// TwinCAT 3 PLC project txi_optics
// Title: lcls-plc-txi-optics
// Company: SLAC
// ProjectVersion: 0.2.0
// ProgramVersion: 3.1.4022.7
// libraries:
//   LCLS General, * (SLAC)
//   PMPS, * (SLAC - LCLS)
//   Tc2_ControllerToolbox, * (Beckhoff Automation GmbH)
//   Tc2_SerialCom, * (Beckhoff Automation GmbH)
//   Tc2_Standard, * (Beckhoff Automation GmbH)
//   Tc2_System, * (Beckhoff Automation GmbH)
//   Tc2_Utilities, * (Beckhoff Automation GmbH)
//   Tc3_Module, * (Beckhoff Automation GmbH)
//   lcls-twincat-motion,4.1.1,SLAC
//   lcls-twincat-optics,0.7.0,SLAC
// project tree:
//   GVLs/ GVL_COM_Buffers.TcGVL, GVL_M1K3.TcGVL, GVL_M1K3_Constants.TcGVL, GVL_M2K3.TcGVL, GVL_M2K3_Constants.TcGVL, GVL_PMPS.TcGVL, GVL_SerialIO.TcGVL
//   Version/ Global_Version.TcGVL
//   / PiezoDriver.TcTTO, PlcTask.TcTTO, SerialIO.TcTTO
//   POUs/ MAIN.TcPOU, PRG_1_PlcTask.TcPOU, PRG_2_PMPS_POST.TcPOU, PRG_MR1K3_SOMS.TcPOU, PRG_MR2K3_SOMS.TcPOU
//   POUs/Serial Comm/ PiezoSerial.TcPOU, P_Serial_Com.TcPOU
// real-time tasks:
//   TASK PlcTask: cycle T#10ms, priority 20, ADS port 350
//   TASK PiezoDriver: cycle T#1ms, priority 3, ADS port 351
//   TASK SerialIO: cycle T#2ms, priority 1, ADS port 352
// motion (NC):
//   TASK NC-Task 1 SAF: cycle T#2ms, priority 4, ADS port 501
//   TASK NC-Task 1 SVB: cycle T#10ms, priority 8, ADS port 511
//   AXIS M1K3-Yup (id 1)
//     General: UnitName=um
//     Dynamic: Acceleration=5050, Deceleration=5050, Jerk=5100500, DelayTime=0.008
//     Velo: Maximum=100
//     OtherSettings: AllowMotionCmdToSlave=true
//     encoder EncType=29
//       EncPara: ScaleFactorNumerator=1, ScaleFactorDenominator=1000, MaxCount=#xffffffff
//         SoftEndMinControl: Enable=true, Range=8900
//         SoftEndMaxControl: Enable=true, Range=122000
//         Inc: RefSoftSyncMask=#x0000ffff
//     drive DrvType=24
//       DrvPara: Inverse=true
//         Analog: VeloReferenz=500
//         TimeComp: TaskDelayCycles=1
//     controller CtrType=3
//       CtrPara: PriorControlFactor=1
//         PosDiffControl: Range=50, Time=0.2
//         PID: PosTn=0.005, PosIOutputLimit=0.0001, PosDOutputLimit=0, PosIDisableWhenMoving=true, DeadBandPosition=0.001
//         Observer: BandWidth=20
//   AXIS M1K3-Ydwn (id 2)
//     General: UnitName=um
//     Dynamic: Acceleration=5050, Deceleration=5050, Jerk=5100500, DelayTime=0.008
//     Velo: Maximum=100
//     OtherSettings: AllowMotionCmdToSlave=true
//     encoder EncType=29
//       EncPara: ScaleFactorNumerator=1, ScaleFactorDenominator=1000, MaxCount=#xffffffff
//         SoftEndMinControl: Enable=true, Range=8395
//         SoftEndMaxControl: Enable=true, Range=122000
//         Inc: RefSoftSyncMask=#x0000ffff
//     drive DrvType=24
//       DrvPara: Inverse=true
//         Analog: VeloReferenz=500
//         TimeComp: TaskDelayCycles=1
//     controller CtrType=3
//       CtrPara: PriorControlFactor=1
//         PosDiffControl: Range=50, Time=0.2
//         PID: PosTn=0.005, PosIOutputLimit=0.0001, PosDOutputLimit=0, PosIDisableWhenMoving=true, DeadBandPosition=0.001
//         Observer: BandWidth=20
//   AXIS M1K3-Xup (id 3)
//     General: UnitName=um
//     Dynamic: AccelerationMaximum=1000, DecelerationMaximum=1000, Acceleration=1000, Deceleration=1000, Jerk=5000, DelayTime=0.008
//     Velo: Maximum=300
//     OtherSettings: AllowMotionCmdToSlave=true
//     encoder EncType=29
//       EncPara: ScaleFactorNumerator=1, ScaleFactorDenominator=1000, MaxCount=#xffffffff
//         SoftEndMinControl: Enable=true, Range=20176
//         SoftEndMaxControl: Enable=true, Range=21576
//         Inc: RefSoftSyncMask=#x0000ffff
//     drive DrvType=24
//       DrvPara: Inverse=true
//         Analog: VeloReferenz=625
//         TimeComp: TaskDelayCycles=1
//     controller CtrType=3
//       CtrPara: PriorControlFactor=1
//         PosDiffControl: Range=50, Time=0.2
//         PID: PosTn=0.005, PosIOutputLimit=0.0001, PosDOutputLimit=0, PosIDisableWhenMoving=true, DeadBandPosition=0.001
//         Observer: BandWidth=20
//   AXIS M1K3-Xdwn (id 4)
//     General: UnitName=um
//     Dynamic: AccelerationMaximum=1000, DecelerationMaximum=1000, Acceleration=1000, Deceleration=1000, Jerk=5000, DelayTime=0.008
//     Velo: Maximum=300
//     OtherSettings: AllowMotionCmdToSlave=true
//     encoder EncType=29
//       EncPara: ScaleFactorNumerator=1, ScaleFactorDenominator=1000, MaxCount=#xffffffff
//         SoftEndMinControl: Enable=true, Range=21276
//         SoftEndMaxControl: Enable=true, Range=22876
//         Inc: RefSoftSyncMask=#x0000ffff
//     drive DrvType=24
//       Analog: VeloReferenz=625
//       TimeComp: TaskDelayCycles=1
//     controller CtrType=3
//       CtrPara: PriorControlFactor=1
//         PosDiffControl: Range=50, Time=0.2
//         PID: PosTn=0.005, PosIOutputLimit=0.0001, PosDOutputLimit=0, PosIDisableWhenMoving=true, DeadBandPosition=0.001
//         Observer: BandWidth=20
//   AXIS M1K3-Pitch (id 5)
//     General: UnitName=urad
//     Dynamic: Acceleration=64082, Deceleration=64082, Jerk=711156, DelayTime=0.008
//     Velo: Maximum=50
//     OtherSettings: AllowMotionCmdToSlave=true
//     encoder EncType=29
//       EncPara: ScaleFactorNumerator=0.00556, MaxCount=#xffffffff
//         SoftEndMinControl: Enable=true, Range=53575
//         SoftEndMaxControl: Enable=true, Range=54180
//         ActPosCorrection: Time=0.008
//         Inc: RefSoftSyncMask=#x0000ffff
//     drive DrvType=24
//       DrvPara: Inverse=true
//         Analog: VeloReferenz=550
//         TimeComp: TaskDelayCycles=1
//     controller CtrType=3
//       CtrPara: PriorControlFactor=1
//         PosDiffControl: Range=10, Time=0.2
//         PID: PosKp=9, PosTn=0.0006, PosTv=1.2e-05, PosIOutputLimit=0.0005, PosDOutputLimit=0.0035, AccKa=0.001, DeadBandPosition=0.1
//         Observer: BandWidth=20
//   AXIS Axis-None1 (id 11)
//     OtherSettings: AllowMotionCmdToSlave=true
//     encoder EncType=1
//     drive DrvType=5
//       Analog: ScaleFactorActTorque=0.1
//     controller CtrType=1
//       CtrPara: PriorControlFactor=1
//         Observer: BandWidth=20
//   AXIS M2K3-Yup (id 6)
//     General: UnitName=um
//     Dynamic: Acceleration=5050, Deceleration=5050, Jerk=5100500, DelayTime=0.008
//     Velo: Maximum=100
//     TargetPosControl: Range=0.05, Time=0.01
//     OtherSettings: AllowMotionCmdToSlave=true
//     encoder EncType=29
//       EncPara: ScaleFactorNumerator=1, ScaleFactorDenominator=1000, MaxCount=#xffffffff
//         SoftEndMinControl: Enable=true, Range=7250
//         SoftEndMaxControl: Enable=true, Range=115658
//         Inc: RefSoftSyncMask=#x0000ffff
//     drive DrvType=24
//       DrvPara: Inverse=true
//         Analog: VeloReferenz=500
//         TimeComp: TaskDelayCycles=1
//     controller CtrType=3
//       CtrPara: PriorControlFactor=1
//         PosDiffControl: Range=50, Time=0.2
//         PID: PosTn=0.005, PosIOutputLimit=0.0001, PosDOutputLimit=0, PosIDisableWhenMoving=true, DeadBandPosition=0.001
//         Observer: BandWidth=20
//   AXIS M2K3-Ydwn (id 7)
//     General: UnitName=um
//     Dynamic: Acceleration=5050, Deceleration=5050, Jerk=5100500, DelayTime=0.008
//     Velo: Maximum=100
//     TargetPosControl: Range=0.05, Time=0.01
//     OtherSettings: AllowMotionCmdToSlave=true
//     encoder EncType=29
//       EncPara: ScaleFactorNumerator=1, ScaleFactorDenominator=1000, MaxCount=#xffffffff
//         SoftEndMinControl: Enable=true, Range=9960
//         SoftEndMaxControl: Enable=true, Range=118260
//         Inc: RefSoftSyncMask=#x0000ffff
//     drive DrvType=24
//       DrvPara: Inverse=true
//         Analog: VeloReferenz=500
//         TimeComp: TaskDelayCycles=1
//     controller CtrType=3
//       CtrPara: PriorControlFactor=1
//         PosDiffControl: Range=50, Time=0.2
//         PID: PosTn=0.005, PosIOutputLimit=0.0001, PosDOutputLimit=0, PosIDisableWhenMoving=true, DeadBandPosition=0.001
//         Observer: BandWidth=20
//   AXIS M2K3-Xup (id 8)
//     General: UnitName=um
//     Dynamic: AccelerationMaximum=1000, DecelerationMaximum=1000, Acceleration=1000, Deceleration=1000, Jerk=5000, DelayTime=0.008
//     Velo: Maximum=150
//     TargetPosControl: Range=0.05, Time=0.01
//     OtherSettings: AllowMotionCmdToSlave=true
//     encoder EncType=29
//       EncPara: ScaleFactorNumerator=1, ScaleFactorDenominator=1000, MaxCount=#xffffffff
//         SoftEndMinControl: Enable=true, Range=19294
//         SoftEndMaxControl: Enable=true, Range=20694
//         Inc: RefSoftSyncMask=#x0000ffff
//     drive DrvType=24
//       DrvPara: Inverse=true
//         Analog: VeloReferenz=625
//         TimeComp: TaskDelayCycles=1
//     controller CtrType=3
//       CtrPara: PriorControlFactor=1
//         PosDiffControl: Range=50, Time=0.2
//         PID: PosTn=0.005, PosIOutputLimit=0.0001, PosDOutputLimit=0, PosIDisableWhenMoving=true, DeadBandPosition=0.001
//         Observer: BandWidth=20
//   AXIS M2K3-Xdwn (id 9)
//     General: UnitName=um
//     Dynamic: AccelerationMaximum=1000, DecelerationMaximum=1000, Acceleration=1000, Deceleration=1000, Jerk=5000, DelayTime=0.008
//     Velo: Maximum=150
//     TargetPosControl: Range=0.05, Time=0.01
//     OtherSettings: AllowMotionCmdToSlave=true
//     encoder EncType=29
//       EncPara: ScaleFactorNumerator=1, ScaleFactorDenominator=1000, MaxCount=#xffffffff
//         SoftEndMinControl: Enable=true, Range=18074
//         SoftEndMaxControl: Enable=true, Range=19674
//         Inc: RefSoftSyncMask=#x0000ffff
//     drive DrvType=24
//       Analog: VeloReferenz=625
//       TimeComp: TaskDelayCycles=1
//     controller CtrType=3
//       CtrPara: PriorControlFactor=1
//         PosDiffControl: Range=50, Time=0.2
//         PID: PosTn=0.005, PosIOutputLimit=0.0001, PosDOutputLimit=0, PosIDisableWhenMoving=true, DeadBandPosition=0.001
//         Observer: BandWidth=20
//   AXIS M2K3-Pitch (id 10)
//     General: UnitName=urad
//     Dynamic: Acceleration=64082, Deceleration=64082, Jerk=711156, DelayTime=0.008
//     Velo: SlowManual=10, FastManual=30, Maximum=50
//     TargetPosControl: Range=0.1, Time=0.01
//     PEHControl: Time=7
//     OtherSettings: AllowMotionCmdToSlave=true
//     encoder EncType=29
//       EncPara: ScaleFactorNumerator=0.00556, MaxCount=#xffffffff
//         FilterTime: TPos=0.05
//         SoftEndMinControl: Enable=true, Range=57450
//         SoftEndMaxControl: Enable=true, Range=59067
//         ActPosCorrection: Time=0.008
//         Inc: RefSoftSyncMask=#x0000ffff
//     drive DrvType=24
//       DrvPara: Inverse=true
//         Analog: VeloReferenz=550
//         TimeComp: TaskDelayCycles=1
//     controller CtrType=3
//       CtrPara: PriorControlFactor=1
//         PosDiffControl: Range=10, Time=0.2
//         PID: PosKp=9, PosTn=0.0006, PosTv=1.2e-05, PosIOutputLimit=0.0005, PosDOutputLimit=0.0035, AccKa=0.001, DeadBandPosition=0.001
//         Observer: BandWidth=20
//   AXIS Axis-None2 (id 12)
//     OtherSettings: AllowMotionCmdToSlave=true
//     encoder EncType=1
//     drive DrvType=5
//       Analog: ScaleFactorActTorque=0.1
//     controller CtrType=1
//       CtrPara: PriorControlFactor=1
//         Observer: BandWidth=20
// I/O:
//   DEVICE Device 1 (EtherCAT), AmsNetId 172.21.88.54.2.1
//     Term 1 (EK1200) [EK1200-5000 EtherCAT Power supply (2A E-Bus)]
//       PMPS_FFO [EL2202 2Ch. Dig. Output 24V, 0.5A]
//       Term 3 (EL6070)
//       PMPS_PRE [EL6695 EtherCAT Bridge terminal (Primary)]
//       Term 6 (EK1122) [EK1122 2 port EtherCAT junction]
//         EK1100_M1K3 [EK1100 EtherCAT Coupler (2A E-Bus)]
//           Term 8 (EL9410)
//           EL7047_M1K3_Yup [EL7047 1Ch. Stepper motor output stage (50V, 5A)]
//           EL7047_M1K3_Ydwn [EL7047 1Ch. Stepper motor output stage (50V, 5A)]
//           EL7047_M1K3_Xup [EL7047 1Ch. Stepper motor output stage (50V, 5A)]
//           EL7047_M1K3_Xdwn [EL7047 1Ch. Stepper motor output stage (50V, 5A)]
//           EL7047_M1K3_PitchCoarse [EL7047 1Ch. Stepper motor output stage (50V, 5A)]
//           EL5042_M1K3_Yupdwn [EL5042 2Ch. BiSS-C Encoder]
//           EL5042_M1K3_Xupdwn
//           EL5042_M1K3_Pitch [EL5042 2Ch. BiSS-C Encoder]
//           EL6001_M1K3_PitchFine [EL6001 Interface (RS232)]
//           EL3054_M1K3_FWM_PRSM [EL3054 4Ch. Ana. Input 4-20mA]
//           Term 19 (EL3202-0010)
//           Term 20 (EL3202-0010)
//           EL1004_M1K3_STO [EL1004 4Ch. Dig. Input 24V, 3ms]
//           EL2004_M1K3_VCV [EL2004 4Ch. Dig. Output 24V, 0.5A]
//           Term 36 (EL9011) [EL9011 End Terminal]
//         EK1100_M2K3 [EK1100 EtherCAT Coupler (2A E-Bus)]
//           Term 22 (EL9410) [EL9410 E-Bus Power Supplier  (Diagnostics)]
//           EL7047_M2K3_Yup [EL7047 1Ch. Stepper motor output stage (50V, 5A)]
//           EL7047_M2K3_Ydwn [EL7047 1Ch. Stepper motor output stage (50V, 5A)]
//           EL7047_M2K3_Xup [EL7047 1Ch. Stepper motor output stage (50V, 5A)]
//           EL7047_M2K3_Xdwn [EL7047 1Ch. Stepper motor output stage (50V, 5A)]
//           EL7047_M2K3_PitchCoarse [EL7047 1Ch. Stepper motor output stage (50V, 5A)]
//           EL5042_M2K3_Yupdwn [EL5042 2Ch. BiSS-C Encoder]
//           EL5042_M2K3_Xupdwn [EL5042 2Ch. BiSS-C Encoder]
//           EL5042_M2K3_Pitch [EL5042 2Ch. BiSS-C Encoder]
//           EL6001_M2K3_PitchFine [EL6001 Interface (RS232)]
//           EL3054_M2K3_FWM_PRSM [EL3054 4Ch. Ana. Input 4-20mA]
//           Term 33 (EL3202-0010) [EL3202-0010 2Ch. Ana. Input PT100 (RTD), High Precision]
//           Term 34 (EL3202-0010) [EL3202-0010 2Ch. Ana. Input PT100 (RTD), High Precision]
//           EL1004_M2K3_STO [EL1004 4Ch. Dig. Input 24V, 3ms]
//           EL2004_M2K3_VCV [EL2004 4Ch. Dig. Output 24V, 0.5A]
//           Term 37 (EL9011) [EL9011 End Terminal]
//       Term 35 (EK1122) [EK1122 2 port EtherCAT junction]
//       Term 38 (EL9011)
// variable links:
//   (this object) <-> Device 1 (EtherCAT)/Term 1 (EK1200)/Term 6 (EK1122)/EK1100_M1K3/EL5042_M1K3_Yupdwn
//     Enc/Inputs/In/nComState @bit 1 <-> WcState/InputToggle
//     Enc/Inputs/In/nComState <-> WcState/WcState
//     Enc/Inputs/In/nDataIn1 <-> FB Inputs Channel 1/Position
//     Enc/Inputs/In/nDataIn1 <-> FB Inputs Channel 2/Position
//     Enc/Inputs/In/nState1 @bit 12 <-> FB Inputs Channel 1/Status/Diag
//     Enc/Inputs/In/nState1 @bit 12 <-> FB Inputs Channel 2/Status/Diag
//     Enc/Inputs/In/nState1 @bit 1 <-> FB Inputs Channel 1/Status/Error
//     Enc/Inputs/In/nState1 @bit 1 <-> FB Inputs Channel 2/Status/Error
//     Enc/Inputs/In/nState1 @bit 14 <-> FB Inputs Channel 1/Status/Input cycle counter
//     Enc/Inputs/In/nState1 @bit 14 <-> FB Inputs Channel 2/Status/Input cycle counter
//     Enc/Inputs/In/nState1 @bit 2 <-> FB Inputs Channel 1/Status/Ready
//     Enc/Inputs/In/nState1 @bit 2 <-> FB Inputs Channel 2/Status/Ready
//     Enc/Inputs/In/nState1 @bit 13 <-> FB Inputs Channel 1/Status/TxPDO State
//     Enc/Inputs/In/nState1 @bit 13 <-> FB Inputs Channel 2/Status/TxPDO State
//     Enc/Inputs/In/nState1 <-> FB Inputs Channel 1/Status/Warning
//     Enc/Inputs/In/nState1 <-> FB Inputs Channel 2/Status/Warning
//   (this object) <-> Device 1 (EtherCAT)/Term 1 (EK1200)/Term 6 (EK1122)/EK1100_M1K3/EL7047_M1K3_Yup
//     Drive/Inputs/In/nState1 @bit 3 <-> STM Status/Status/Error
//     Drive/Inputs/In/nState1 @bit 7 <-> STM Status/Status/Motor stall
//     Drive/Inputs/In/nState1 @bit 5 <-> STM Status/Status/Moving negative
//     Drive/Inputs/In/nState1 @bit 4 <-> STM Status/Status/Moving positive
//     Drive/Inputs/In/nState1 @bit 1 <-> STM Status/Status/Ready
//     Drive/Inputs/In/nState1 <-> STM Status/Status/Ready to enable
//     Drive/Inputs/In/nState1 @bit 6 <-> STM Status/Status/Torque reduced
//     Drive/Inputs/In/nState1 @bit 2 <-> STM Status/Status/Warning
//     Drive/Inputs/In/nState2 @bit 3 <-> STM Status/Status/Digital input 1
//     Drive/Inputs/In/nState2 @bit 4 <-> STM Status/Status/Digital input 2
//     Drive/Inputs/In/nState2 @bit 5 <-> STM Status/Status/Sync error
//     Drive/Inputs/In/nState2 @bit 7 <-> STM Status/Status/TxPDO Toggle
//     Drive/Inputs/In/nState4 @bit 1 <-> WcState/InputToggle
//     Drive/Inputs/In/nState4 <-> WcState/WcState
//     Drive/Outputs/Out/nCtrl1 <-> STM Control/Control/Enable
//     Drive/Outputs/Out/nCtrl1 @bit 2 <-> STM Control/Control/Reduce torque
//     Drive/Outputs/Out/nCtrl1 @bit 1 <-> STM Control/Control/Reset
//     Drive/Outputs/Out/nCtrl2 @bit 3 <-> STM Control/Control/Digital output 1
//     Drive/Outputs/Out/nDataOut2[0] <-> STM Velocity/Velocity
//   (this object) <-> Device 1 (EtherCAT)/Term 1 (EK1200)/Term 6 (EK1122)/EK1100_M1K3/EL7047_M1K3_Ydwn
//     Drive/Inputs/In/nState1 @bit 3 <-> STM Status/Status/Error
//     Drive/Inputs/In/nState1 @bit 7 <-> STM Status/Status/Motor stall
//     Drive/Inputs/In/nState1 @bit 5 <-> STM Status/Status/Moving negative
//     Drive/Inputs/In/nState1 @bit 4 <-> STM Status/Status/Moving positive
//     Drive/Inputs/In/nState1 @bit 1 <-> STM Status/Status/Ready
//     Drive/Inputs/In/nState1 <-> STM Status/Status/Ready to enable
//     Drive/Inputs/In/nState1 @bit 6 <-> STM Status/Status/Torque reduced
//     Drive/Inputs/In/nState1 @bit 2 <-> STM Status/Status/Warning
//     Drive/Inputs/In/nState2 @bit 3 <-> STM Status/Status/Digital input 1
//     Drive/Inputs/In/nState2 @bit 4 <-> STM Status/Status/Digital input 2
//     Drive/Inputs/In/nState2 @bit 5 <-> STM Status/Status/Sync error
//     Drive/Inputs/In/nState2 @bit 7 <-> STM Status/Status/TxPDO Toggle
//     Drive/Inputs/In/nState4 @bit 1 <-> WcState/InputToggle
//     Drive/Inputs/In/nState4 <-> WcState/WcState
//     Drive/Outputs/Out/nCtrl1 <-> STM Control/Control/Enable
//     Drive/Outputs/Out/nCtrl1 @bit 2 <-> STM Control/Control/Reduce torque
//     Drive/Outputs/Out/nCtrl1 @bit 1 <-> STM Control/Control/Reset
//     Drive/Outputs/Out/nCtrl2 @bit 3 <-> STM Control/Control/Digital output 1
//     Drive/Outputs/Out/nDataOut2[0] <-> STM Velocity/Velocity
//   (this object) <-> Device 1 (EtherCAT)/Term 1 (EK1200)/Term 6 (EK1122)/EK1100_M1K3/EL5042_M1K3_Xupdwn
//     Enc/Inputs/In/nComState @bit 1 <-> WcState/InputToggle
//     Enc/Inputs/In/nComState <-> WcState/WcState
//     Enc/Inputs/In/nDataIn1 <-> FB Inputs Channel 1/Position
//     Enc/Inputs/In/nDataIn1 <-> FB Inputs Channel 2/Position
//     Enc/Inputs/In/nState1 @bit 12 <-> FB Inputs Channel 1/Status/Diag
//     Enc/Inputs/In/nState1 @bit 12 <-> FB Inputs Channel 2/Status/Diag
//     Enc/Inputs/In/nState1 @bit 1 <-> FB Inputs Channel 1/Status/Error
//     Enc/Inputs/In/nState1 @bit 1 <-> FB Inputs Channel 2/Status/Error
//     Enc/Inputs/In/nState1 @bit 14 <-> FB Inputs Channel 1/Status/Input cycle counter
//     Enc/Inputs/In/nState1 @bit 14 <-> FB Inputs Channel 2/Status/Input cycle counter
//     Enc/Inputs/In/nState1 @bit 2 <-> FB Inputs Channel 1/Status/Ready
//     Enc/Inputs/In/nState1 @bit 2 <-> FB Inputs Channel 2/Status/Ready
//     Enc/Inputs/In/nState1 @bit 13 <-> FB Inputs Channel 1/Status/TxPDO State
//     Enc/Inputs/In/nState1 @bit 13 <-> FB Inputs Channel 2/Status/TxPDO State
//     Enc/Inputs/In/nState1 <-> FB Inputs Channel 1/Status/Warning
//     Enc/Inputs/In/nState1 <-> FB Inputs Channel 2/Status/Warning
//   (this object) <-> Device 1 (EtherCAT)/Term 1 (EK1200)/Term 6 (EK1122)/EK1100_M1K3/EL7047_M1K3_Xup
//     Drive/Inputs/In/nState1 @bit 3 <-> STM Status/Status/Error
//     Drive/Inputs/In/nState1 @bit 7 <-> STM Status/Status/Motor stall
//     Drive/Inputs/In/nState1 @bit 5 <-> STM Status/Status/Moving negative
//     Drive/Inputs/In/nState1 @bit 4 <-> STM Status/Status/Moving positive
//     Drive/Inputs/In/nState1 @bit 1 <-> STM Status/Status/Ready
//     Drive/Inputs/In/nState1 <-> STM Status/Status/Ready to enable
//     Drive/Inputs/In/nState1 @bit 6 <-> STM Status/Status/Torque reduced
//     Drive/Inputs/In/nState1 @bit 2 <-> STM Status/Status/Warning
//     Drive/Inputs/In/nState2 @bit 3 <-> STM Status/Status/Digital input 1
//     Drive/Inputs/In/nState2 @bit 4 <-> STM Status/Status/Digital input 2
//     Drive/Inputs/In/nState2 @bit 5 <-> STM Status/Status/Sync error
//     Drive/Inputs/In/nState2 @bit 7 <-> STM Status/Status/TxPDO Toggle
//     Drive/Inputs/In/nState4 @bit 1 <-> WcState/InputToggle
//     Drive/Inputs/In/nState4 <-> WcState/WcState
//     Drive/Outputs/Out/nCtrl1 <-> STM Control/Control/Enable
//     Drive/Outputs/Out/nCtrl1 @bit 2 <-> STM Control/Control/Reduce torque
//     Drive/Outputs/Out/nCtrl1 @bit 1 <-> STM Control/Control/Reset
//     Drive/Outputs/Out/nCtrl2 @bit 3 <-> STM Control/Control/Digital output 1
//     Drive/Outputs/Out/nDataOut2[0] <-> STM Velocity/Velocity
//   (this object) <-> Device 1 (EtherCAT)/Term 1 (EK1200)/Term 6 (EK1122)/EK1100_M1K3/EL7047_M1K3_Xdwn
//     Drive/Inputs/In/nState1 @bit 3 <-> STM Status/Status/Error
//     Drive/Inputs/In/nState1 @bit 7 <-> STM Status/Status/Motor stall
//     Drive/Inputs/In/nState1 @bit 5 <-> STM Status/Status/Moving negative
//     Drive/Inputs/In/nState1 @bit 4 <-> STM Status/Status/Moving positive
//     Drive/Inputs/In/nState1 @bit 1 <-> STM Status/Status/Ready
//     Drive/Inputs/In/nState1 <-> STM Status/Status/Ready to enable
//     Drive/Inputs/In/nState1 @bit 6 <-> STM Status/Status/Torque reduced
//     Drive/Inputs/In/nState1 @bit 2 <-> STM Status/Status/Warning
//     Drive/Inputs/In/nState2 @bit 3 <-> STM Status/Status/Digital input 1
//     Drive/Inputs/In/nState2 @bit 4 <-> STM Status/Status/Digital input 2
//     Drive/Inputs/In/nState2 @bit 5 <-> STM Status/Status/Sync error
//     Drive/Inputs/In/nState2 @bit 7 <-> STM Status/Status/TxPDO Toggle
//     Drive/Inputs/In/nState4 @bit 1 <-> WcState/InputToggle
//     Drive/Inputs/In/nState4 <-> WcState/WcState
//     Drive/Outputs/Out/nCtrl1 <-> STM Control/Control/Enable
//     Drive/Outputs/Out/nCtrl1 @bit 2 <-> STM Control/Control/Reduce torque
//     Drive/Outputs/Out/nCtrl1 @bit 1 <-> STM Control/Control/Reset
//     Drive/Outputs/Out/nCtrl2 @bit 3 <-> STM Control/Control/Digital output 1
//     Drive/Outputs/Out/nDataOut2[0] <-> STM Velocity/Velocity
//   (this object) <-> Device 1 (EtherCAT)/Term 1 (EK1200)/Term 6 (EK1122)/EK1100_M1K3/EL5042_M1K3_Pitch
//     Enc/Inputs/In/nComState @bit 1 <-> WcState/InputToggle
//     Enc/Inputs/In/nComState <-> WcState/WcState
//     Enc/Inputs/In/nDataIn1 <-> FB Inputs Channel 1/Position
//     Enc/Inputs/In/nState1 @bit 12 <-> FB Inputs Channel 1/Status/Diag
//     Enc/Inputs/In/nState1 @bit 1 <-> FB Inputs Channel 1/Status/Error
//     Enc/Inputs/In/nState1 @bit 14 <-> FB Inputs Channel 1/Status/Input cycle counter
//     Enc/Inputs/In/nState1 @bit 2 <-> FB Inputs Channel 1/Status/Ready
//     Enc/Inputs/In/nState1 @bit 13 <-> FB Inputs Channel 1/Status/TxPDO State
//     Enc/Inputs/In/nState1 <-> FB Inputs Channel 1/Status/Warning
//   (this object) <-> Device 1 (EtherCAT)/Term 1 (EK1200)/Term 6 (EK1122)/EK1100_M1K3/EL7047_M1K3_PitchCoarse
//     Drive/Inputs/In/nState1 @bit 3 <-> STM Status/Status/Error
//     Drive/Inputs/In/nState1 @bit 7 <-> STM Status/Status/Motor stall
//     Drive/Inputs/In/nState1 @bit 5 <-> STM Status/Status/Moving negative
//     Drive/Inputs/In/nState1 @bit 4 <-> STM Status/Status/Moving positive
//     Drive/Inputs/In/nState1 @bit 1 <-> STM Status/Status/Ready
//     Drive/Inputs/In/nState1 <-> STM Status/Status/Ready to enable
//     Drive/Inputs/In/nState1 @bit 6 <-> STM Status/Status/Torque reduced
//     Drive/Inputs/In/nState1 @bit 2 <-> STM Status/Status/Warning
//     Drive/Inputs/In/nState2 @bit 3 <-> STM Status/Status/Digital input 1
//     Drive/Inputs/In/nState2 @bit 4 <-> STM Status/Status/Digital input 2
//     Drive/Inputs/In/nState2 @bit 5 <-> STM Status/Status/Sync error
//     Drive/Inputs/In/nState2 @bit 7 <-> STM Status/Status/TxPDO Toggle
//     Drive/Inputs/In/nState4 @bit 1 <-> WcState/InputToggle
//     Drive/Inputs/In/nState4 <-> WcState/WcState
//     Drive/Outputs/Out/nCtrl1 <-> STM Control/Control/Enable
//     Drive/Outputs/Out/nCtrl1 @bit 2 <-> STM Control/Control/Reduce torque
//     Drive/Outputs/Out/nCtrl1 @bit 1 <-> STM Control/Control/Reset
//     Drive/Outputs/Out/nCtrl2 @bit 3 <-> STM Control/Control/Digital output 1
//     Drive/Outputs/Out/nDataOut2[0] <-> STM Velocity/Velocity
//   (this object) <-> Device 1 (EtherCAT)/Term 1 (EK1200)/Term 6 (EK1122)/EK1100_M2K3/EL5042_M2K3_Yupdwn
//     Enc/Inputs/In/nComState @bit 1 <-> WcState/InputToggle
//     Enc/Inputs/In/nComState <-> WcState/WcState
//     Enc/Inputs/In/nDataIn1 <-> FB Inputs Channel 1/Position
//     Enc/Inputs/In/nDataIn1 <-> FB Inputs Channel 2/Position
//     Enc/Inputs/In/nState1 @bit 12 <-> FB Inputs Channel 1/Status/Diag
//     Enc/Inputs/In/nState1 @bit 12 <-> FB Inputs Channel 2/Status/Diag
//     Enc/Inputs/In/nState1 @bit 1 <-> FB Inputs Channel 1/Status/Error
//     Enc/Inputs/In/nState1 @bit 1 <-> FB Inputs Channel 2/Status/Error
//     Enc/Inputs/In/nState1 @bit 14 <-> FB Inputs Channel 1/Status/Input cycle counter
//     Enc/Inputs/In/nState1 @bit 14 <-> FB Inputs Channel 2/Status/Input cycle counter
//     Enc/Inputs/In/nState1 @bit 2 <-> FB Inputs Channel 1/Status/Ready
//     Enc/Inputs/In/nState1 @bit 2 <-> FB Inputs Channel 2/Status/Ready
//     Enc/Inputs/In/nState1 @bit 13 <-> FB Inputs Channel 1/Status/TxPDO State
//     Enc/Inputs/In/nState1 @bit 13 <-> FB Inputs Channel 2/Status/TxPDO State
//     Enc/Inputs/In/nState1 <-> FB Inputs Channel 1/Status/Warning
//     Enc/Inputs/In/nState1 <-> FB Inputs Channel 2/Status/Warning
//   (this object) <-> Device 1 (EtherCAT)/Term 1 (EK1200)/Term 6 (EK1122)/EK1100_M2K3/EL7047_M2K3_Yup
//     Drive/Inputs/In/nState1 @bit 3 <-> STM Status/Status/Error
//     Drive/Inputs/In/nState1 @bit 7 <-> STM Status/Status/Motor stall
//     Drive/Inputs/In/nState1 @bit 5 <-> STM Status/Status/Moving negative
//     Drive/Inputs/In/nState1 @bit 4 <-> STM Status/Status/Moving positive
//     Drive/Inputs/In/nState1 @bit 1 <-> STM Status/Status/Ready
//     Drive/Inputs/In/nState1 <-> STM Status/Status/Ready to enable
//     Drive/Inputs/In/nState1 @bit 6 <-> STM Status/Status/Torque reduced
//     Drive/Inputs/In/nState1 @bit 2 <-> STM Status/Status/Warning
//     Drive/Inputs/In/nState2 @bit 3 <-> STM Status/Status/Digital input 1
//     Drive/Inputs/In/nState2 @bit 4 <-> STM Status/Status/Digital input 2
//     Drive/Inputs/In/nState2 @bit 5 <-> STM Status/Status/Sync error
//     Drive/Inputs/In/nState2 @bit 7 <-> STM Status/Status/TxPDO Toggle
//     Drive/Inputs/In/nState4 @bit 1 <-> WcState/InputToggle
//     Drive/Inputs/In/nState4 <-> WcState/WcState
//     Drive/Outputs/Out/nCtrl1 <-> STM Control/Control/Enable
//     Drive/Outputs/Out/nCtrl1 @bit 2 <-> STM Control/Control/Reduce torque
//     Drive/Outputs/Out/nCtrl1 @bit 1 <-> STM Control/Control/Reset
//     Drive/Outputs/Out/nCtrl2 @bit 3 <-> STM Control/Control/Digital output 1
//     Drive/Outputs/Out/nDataOut2[0] <-> STM Velocity/Velocity
//   (this object) <-> Device 1 (EtherCAT)/Term 1 (EK1200)/Term 6 (EK1122)/EK1100_M2K3/EL7047_M2K3_Ydwn
//     Drive/Inputs/In/nState1 @bit 3 <-> STM Status/Status/Error
//     Drive/Inputs/In/nState1 @bit 7 <-> STM Status/Status/Motor stall
//     Drive/Inputs/In/nState1 @bit 5 <-> STM Status/Status/Moving negative
//     Drive/Inputs/In/nState1 @bit 4 <-> STM Status/Status/Moving positive
//     Drive/Inputs/In/nState1 @bit 1 <-> STM Status/Status/Ready
//     Drive/Inputs/In/nState1 <-> STM Status/Status/Ready to enable
//     Drive/Inputs/In/nState1 @bit 6 <-> STM Status/Status/Torque reduced
//     Drive/Inputs/In/nState1 @bit 2 <-> STM Status/Status/Warning
//     Drive/Inputs/In/nState2 @bit 3 <-> STM Status/Status/Digital input 1
//     Drive/Inputs/In/nState2 @bit 4 <-> STM Status/Status/Digital input 2
//     Drive/Inputs/In/nState2 @bit 5 <-> STM Status/Status/Sync error
//     Drive/Inputs/In/nState2 @bit 7 <-> STM Status/Status/TxPDO Toggle
//     Drive/Inputs/In/nState4 @bit 1 <-> WcState/InputToggle
//     Drive/Inputs/In/nState4 <-> WcState/WcState
//     Drive/Outputs/Out/nCtrl1 <-> STM Control/Control/Enable
//     Drive/Outputs/Out/nCtrl1 @bit 2 <-> STM Control/Control/Reduce torque
//     Drive/Outputs/Out/nCtrl1 @bit 1 <-> STM Control/Control/Reset
//     Drive/Outputs/Out/nCtrl2 @bit 3 <-> STM Control/Control/Digital output 1
//     Drive/Outputs/Out/nDataOut2[0] <-> STM Velocity/Velocity
//   (this object) <-> Device 1 (EtherCAT)/Term 1 (EK1200)/Term 6 (EK1122)/EK1100_M2K3/EL5042_M2K3_Xupdwn
//     Enc/Inputs/In/nComState @bit 1 <-> WcState/InputToggle
//     Enc/Inputs/In/nComState <-> WcState/WcState
//     Enc/Inputs/In/nDataIn1 <-> FB Inputs Channel 1/Position
//     Enc/Inputs/In/nDataIn1 <-> FB Inputs Channel 2/Position
//     Enc/Inputs/In/nState1 @bit 12 <-> FB Inputs Channel 1/Status/Diag
//     Enc/Inputs/In/nState1 @bit 12 <-> FB Inputs Channel 2/Status/Diag
//     Enc/Inputs/In/nState1 @bit 1 <-> FB Inputs Channel 1/Status/Error
//     Enc/Inputs/In/nState1 @bit 1 <-> FB Inputs Channel 2/Status/Error
//     Enc/Inputs/In/nState1 @bit 14 <-> FB Inputs Channel 1/Status/Input cycle counter
//     Enc/Inputs/In/nState1 @bit 14 <-> FB Inputs Channel 2/Status/Input cycle counter
//     Enc/Inputs/In/nState1 @bit 2 <-> FB Inputs Channel 1/Status/Ready
//     Enc/Inputs/In/nState1 @bit 2 <-> FB Inputs Channel 2/Status/Ready
//     Enc/Inputs/In/nState1 @bit 13 <-> FB Inputs Channel 1/Status/TxPDO State
//     Enc/Inputs/In/nState1 @bit 13 <-> FB Inputs Channel 2/Status/TxPDO State
//     Enc/Inputs/In/nState1 <-> FB Inputs Channel 1/Status/Warning
//     Enc/Inputs/In/nState1 <-> FB Inputs Channel 2/Status/Warning
//   (this object) <-> Device 1 (EtherCAT)/Term 1 (EK1200)/Term 6 (EK1122)/EK1100_M2K3/EL7047_M2K3_Xup
//     Drive/Inputs/In/nState1 @bit 3 <-> STM Status/Status/Error
//     Drive/Inputs/In/nState1 @bit 7 <-> STM Status/Status/Motor stall
//     Drive/Inputs/In/nState1 @bit 5 <-> STM Status/Status/Moving negative
//     Drive/Inputs/In/nState1 @bit 4 <-> STM Status/Status/Moving positive
//     Drive/Inputs/In/nState1 @bit 1 <-> STM Status/Status/Ready
//     Drive/Inputs/In/nState1 <-> STM Status/Status/Ready to enable
//     Drive/Inputs/In/nState1 @bit 6 <-> STM Status/Status/Torque reduced
//     Drive/Inputs/In/nState1 @bit 2 <-> STM Status/Status/Warning
//     Drive/Inputs/In/nState2 @bit 3 <-> STM Status/Status/Digital input 1
//     Drive/Inputs/In/nState2 @bit 4 <-> STM Status/Status/Digital input 2
//     Drive/Inputs/In/nState2 @bit 5 <-> STM Status/Status/Sync error
//     Drive/Inputs/In/nState2 @bit 7 <-> STM Status/Status/TxPDO Toggle
//     Drive/Inputs/In/nState4 @bit 1 <-> WcState/InputToggle
//     Drive/Inputs/In/nState4 <-> WcState/WcState
//     Drive/Outputs/Out/nCtrl1 <-> STM Control/Control/Enable
//     Drive/Outputs/Out/nCtrl1 @bit 2 <-> STM Control/Control/Reduce torque
//     Drive/Outputs/Out/nCtrl1 @bit 1 <-> STM Control/Control/Reset
//     Drive/Outputs/Out/nCtrl2 @bit 3 <-> STM Control/Control/Digital output 1
//     Drive/Outputs/Out/nDataOut2[0] <-> STM Velocity/Velocity
//   (this object) <-> Device 1 (EtherCAT)/Term 1 (EK1200)/Term 6 (EK1122)/EK1100_M2K3/EL7047_M2K3_Xdwn
//     Drive/Inputs/In/nState1 @bit 3 <-> STM Status/Status/Error
//     Drive/Inputs/In/nState1 @bit 7 <-> STM Status/Status/Motor stall
//     Drive/Inputs/In/nState1 @bit 5 <-> STM Status/Status/Moving negative
//     Drive/Inputs/In/nState1 @bit 4 <-> STM Status/Status/Moving positive
//     Drive/Inputs/In/nState1 @bit 1 <-> STM Status/Status/Ready
//     Drive/Inputs/In/nState1 <-> STM Status/Status/Ready to enable
//     Drive/Inputs/In/nState1 @bit 6 <-> STM Status/Status/Torque reduced
//     Drive/Inputs/In/nState1 @bit 2 <-> STM Status/Status/Warning
//     Drive/Inputs/In/nState2 @bit 3 <-> STM Status/Status/Digital input 1
//     Drive/Inputs/In/nState2 @bit 4 <-> STM Status/Status/Digital input 2
//     Drive/Inputs/In/nState2 @bit 5 <-> STM Status/Status/Sync error
//     Drive/Inputs/In/nState2 @bit 7 <-> STM Status/Status/TxPDO Toggle
//     Drive/Inputs/In/nState4 @bit 1 <-> WcState/InputToggle
//     Drive/Inputs/In/nState4 <-> WcState/WcState
//     Drive/Outputs/Out/nCtrl1 <-> STM Control/Control/Enable
//     Drive/Outputs/Out/nCtrl1 @bit 2 <-> STM Control/Control/Reduce torque
//     Drive/Outputs/Out/nCtrl1 @bit 1 <-> STM Control/Control/Reset
//     Drive/Outputs/Out/nCtrl2 @bit 3 <-> STM Control/Control/Digital output 1
//     Drive/Outputs/Out/nDataOut2[0] <-> STM Velocity/Velocity
//   (this object) <-> Device 1 (EtherCAT)/Term 1 (EK1200)/Term 6 (EK1122)/EK1100_M2K3/EL5042_M2K3_Pitch
//     Enc/Inputs/In/nComState @bit 1 <-> WcState/InputToggle
//     Enc/Inputs/In/nComState <-> WcState/WcState
//     Enc/Inputs/In/nDataIn1 <-> FB Inputs Channel 1/Position
//     Enc/Inputs/In/nState1 @bit 12 <-> FB Inputs Channel 1/Status/Diag
//     Enc/Inputs/In/nState1 @bit 1 <-> FB Inputs Channel 1/Status/Error
//     Enc/Inputs/In/nState1 @bit 14 <-> FB Inputs Channel 1/Status/Input cycle counter
//     Enc/Inputs/In/nState1 @bit 2 <-> FB Inputs Channel 1/Status/Ready
//     Enc/Inputs/In/nState1 @bit 13 <-> FB Inputs Channel 1/Status/TxPDO State
//     Enc/Inputs/In/nState1 <-> FB Inputs Channel 1/Status/Warning
//   (this object) <-> Device 1 (EtherCAT)/Term 1 (EK1200)/Term 6 (EK1122)/EK1100_M2K3/EL7047_M2K3_PitchCoarse
//     Drive/Inputs/In/nState1 @bit 3 <-> STM Status/Status/Error
//     Drive/Inputs/In/nState1 @bit 7 <-> STM Status/Status/Motor stall
//     Drive/Inputs/In/nState1 @bit 5 <-> STM Status/Status/Moving negative
//     Drive/Inputs/In/nState1 @bit 4 <-> STM Status/Status/Moving positive
//     Drive/Inputs/In/nState1 @bit 1 <-> STM Status/Status/Ready
//     Drive/Inputs/In/nState1 <-> STM Status/Status/Ready to enable
//     Drive/Inputs/In/nState1 @bit 6 <-> STM Status/Status/Torque reduced
//     Drive/Inputs/In/nState1 @bit 2 <-> STM Status/Status/Warning
//     Drive/Inputs/In/nState2 @bit 3 <-> STM Status/Status/Digital input 1
//     Drive/Inputs/In/nState2 @bit 4 <-> STM Status/Status/Digital input 2
//     Drive/Inputs/In/nState2 @bit 5 <-> STM Status/Status/Sync error
//     Drive/Inputs/In/nState2 @bit 7 <-> STM Status/Status/TxPDO Toggle
//     Drive/Inputs/In/nState4 @bit 1 <-> WcState/InputToggle
//     Drive/Inputs/In/nState4 <-> WcState/WcState
//     Drive/Outputs/Out/nCtrl1 <-> STM Control/Control/Enable
//     Drive/Outputs/Out/nCtrl1 @bit 2 <-> STM Control/Control/Reduce torque
//     Drive/Outputs/Out/nCtrl1 @bit 1 <-> STM Control/Control/Reset
//     Drive/Outputs/Out/nCtrl2 @bit 3 <-> STM Control/Control/Digital output 1
//     Drive/Outputs/Out/nDataOut2[0] <-> STM Velocity/Velocity
//   txi_optics Instance <-> Device 1 (EtherCAT)/Term 1 (EK1200)/PMPS_PRE
//     PlcTask Inputs/PRG_2_PMPS_POST.fbArbiterIO.i_stCurrentBP <-> IO Inputs/CurrentBP
//     PlcTask Inputs/PRG_2_PMPS_POST.fbArbiterIO.xTxPDO_state <-> SYNC Inputs/TxPDO state
//     PlcTask Inputs/PRG_2_PMPS_POST.fbArbiterIO.xTxPDO_toggle <-> SYNC Inputs/TxPDO toggle
//     PlcTask Outputs/GVL_PMPS.fbFastFaultOutput1.q_xFastFaultOut <-> IO Outputs/FFO
//     PlcTask Outputs/PRG_2_PMPS_POST.fbArbiterIO.q_stRequestedBP <-> IO Outputs/RequestedBP
//     PlcTask Outputs/PRG_MR1K3_SOMS.nMR1K3_Y_ENC_PMPS <-> IO Outputs/MR1K3_Y_ENC
//     PlcTask Outputs/PRG_MR2K3_SOMS.nMR2K3_Y_ENC_PMPS <-> IO Outputs/MR2K3_Y_ENC
//   txi_optics Instance <-> Device 1 (EtherCAT)/Term 1 (EK1200)/Term 6 (EK1122)/EK1100_M1K3/EL1004_M1K3_STO
//     PlcTask Inputs/MAIN.M1K3.fbRunHOMS.bSTOEnable1 <-> Channel 1/Input
//     PlcTask Inputs/MAIN.M1K3.fbRunHOMS.bSTOEnable2 <-> Channel 2/Input
//   txi_optics Instance <-> Device 1 (EtherCAT)/Term 1 (EK1200)/Term 6 (EK1122)/EK1100_M1K3/EL2004_M1K3_VCV
//     PlcTask Outputs/MAIN.bActivateVarCoolMR1K3 <-> Channel 1/Output
//   txi_optics Instance <-> Device 1 (EtherCAT)/Term 1 (EK1200)/Term 6 (EK1122)/EK1100_M1K3/EL3054_M1K3_FWM_PRSM
//     PlcTask Inputs/MAIN.fbCoolingPanelMR1K3.fbFlow_1.iRaw <-> AI Standard Channel 1/Value
//     PlcTask Inputs/MAIN.fbCoolingPanelMR1K3.fbFlow_2.iRaw <-> AI Standard Channel 2/Value
//     PlcTask Inputs/MAIN.fbCoolingPanelMR1K3.fbPress_1.iRaw <-> AI Standard Channel 3/Value
//   txi_optics Instance <-> Device 1 (EtherCAT)/Term 1 (EK1200)/Term 6 (EK1122)/EK1100_M1K3/EL5042_M1K3_Pitch
//     PlcTask Inputs/GVL_M1K3.M1K3_Pitch.diEncCnt <-> FB Inputs Channel 1/Position
//     PlcTask Inputs/MAIN.M5.nRawEncoderULINT <-> FB Inputs Channel 1/Position
//   txi_optics Instance <-> Device 1 (EtherCAT)/Term 1 (EK1200)/Term 6 (EK1122)/EK1100_M1K3/EL5042_M1K3_Xupdwn
//     PlcTask Inputs/MAIN.M1K3.fbRunHOMS.stXdwnEnc/Count <-> FB Inputs Channel 2/Position
//     PlcTask Inputs/MAIN.M1K3.fbRunHOMS.stXupEnc/Count <-> FB Inputs Channel 1/Position
//     PlcTask Inputs/MAIN.M3.nRawEncoderULINT <-> FB Inputs Channel 1/Position
//     PlcTask Inputs/MAIN.M4.nRawEncoderULINT <-> FB Inputs Channel 2/Position
//   txi_optics Instance <-> Device 1 (EtherCAT)/Term 1 (EK1200)/Term 6 (EK1122)/EK1100_M1K3/EL5042_M1K3_Yupdwn
//     PlcTask Inputs/MAIN.M1.nRawEncoderULINT <-> FB Inputs Channel 1/Position
//     PlcTask Inputs/MAIN.M1K3.fbRunHOMS.stYdwnEnc/Count <-> FB Inputs Channel 2/Position
//     PlcTask Inputs/MAIN.M1K3.fbRunHOMS.stYupEnc/Count <-> FB Inputs Channel 1/Position
//     PlcTask Inputs/PRG_MR1K3_SOMS.bMR1K3_Y_ENC_Ready <-> FB Inputs Channel 1/Status/Ready
//     PlcTask Inputs/PRG_MR1K3_SOMS.bMR1K3_Y_ENC_TxPDO <-> FB Inputs Channel 1/Status/TxPDO State
//   txi_optics Instance <-> Device 1 (EtherCAT)/Term 1 (EK1200)/Term 6 (EK1122)/EK1100_M1K3/EL6001_M1K3_PitchFine
//     SerialIO Inputs/GVL_SerialIO.Serial_stComIn_M1K3/D[{0..21}] <-> COM Inputs/Data In {0..21}  (22 links)
//     SerialIO Inputs/GVL_SerialIO.Serial_stComIn_M1K3/Status <-> COM Inputs/Status
//     SerialIO Outputs/GVL_SerialIO.Serial_stComOut_M1K3/Ctrl <-> COM Outputs/Ctrl
//     SerialIO Outputs/GVL_SerialIO.Serial_stComOut_M1K3/D[{0..21}] <-> COM Outputs/Data Out {0..21}  (22 links)
//   txi_optics Instance <-> Device 1 (EtherCAT)/Term 1 (EK1200)/Term 6 (EK1122)/EK1100_M1K3/EL7047_M1K3_PitchCoarse
//     PlcTask Inputs/MAIN.M5.bLimitBackwardEnable <-> STM Status/Status/Digital input 2
//     PlcTask Inputs/MAIN.M5.bLimitForwardEnable <-> STM Status/Status/Digital input 1
//   txi_optics Instance <-> Device 1 (EtherCAT)/Term 1 (EK1200)/Term 6 (EK1122)/EK1100_M1K3/EL7047_M1K3_Xdwn
//     PlcTask Inputs/MAIN.M4.bLimitBackwardEnable <-> STM Status/Status/Digital input 2
//     PlcTask Inputs/MAIN.M4.bLimitForwardEnable <-> STM Status/Status/Digital input 1
//   txi_optics Instance <-> Device 1 (EtherCAT)/Term 1 (EK1200)/Term 6 (EK1122)/EK1100_M1K3/EL7047_M1K3_Xup
//     PlcTask Inputs/MAIN.M3.bLimitBackwardEnable <-> STM Status/Status/Digital input 2
//     PlcTask Inputs/MAIN.M3.bLimitForwardEnable <-> STM Status/Status/Digital input 1
//   txi_optics Instance <-> Device 1 (EtherCAT)/Term 1 (EK1200)/Term 6 (EK1122)/EK1100_M1K3/EL7047_M1K3_Ydwn
//     PlcTask Inputs/MAIN.M2.bLimitBackwardEnable <-> STM Status/Status/Digital input 2
//     PlcTask Inputs/MAIN.M2.bLimitForwardEnable <-> STM Status/Status/Digital input 1
//   txi_optics Instance <-> Device 1 (EtherCAT)/Term 1 (EK1200)/Term 6 (EK1122)/EK1100_M1K3/EL7047_M1K3_Yup
//     PlcTask Inputs/MAIN.M1.bLimitBackwardEnable <-> STM Status/Status/Digital input 2
//     PlcTask Inputs/MAIN.M1.bLimitForwardEnable <-> STM Status/Status/Digital input 1
//   txi_optics Instance <-> Device 1 (EtherCAT)/Term 1 (EK1200)/Term 6 (EK1122)/EK1100_M2K3/EL1004_M2K3_STO
//     PlcTask Inputs/MAIN.M2K3.fbRunHOMS.bSTOEnable1 <-> Channel 1/Input
//     PlcTask Inputs/MAIN.M2K3.fbRunHOMS.bSTOEnable2 <-> Channel 2/Input
//   txi_optics Instance <-> Device 1 (EtherCAT)/Term 1 (EK1200)/Term 6 (EK1122)/EK1100_M2K3/EL2004_M2K3_VCV
//     PlcTask Outputs/MAIN.bActivateVarCoolMR2K3 <-> Channel 1/Output
//   txi_optics Instance <-> Device 1 (EtherCAT)/Term 1 (EK1200)/Term 6 (EK1122)/EK1100_M2K3/EL3054_M2K3_FWM_PRSM
//     PlcTask Inputs/MAIN.fbCoolingPanelMR2K3.fbFlow_1.iRaw <-> AI Standard Channel 1/Value
//     PlcTask Inputs/MAIN.fbCoolingPanelMR2K3.fbFlow_2.iRaw <-> AI Standard Channel 2/Value
//     PlcTask Inputs/MAIN.fbCoolingPanelMR2K3.fbPress_1.iRaw <-> AI Standard Channel 3/Value
//   txi_optics Instance <-> Device 1 (EtherCAT)/Term 1 (EK1200)/Term 6 (EK1122)/EK1100_M2K3/EL5042_M2K3_Pitch
//     PlcTask Inputs/GVL_M2K3.M2K3_Pitch.diEncCnt <-> FB Inputs Channel 1/Position
//     PlcTask Inputs/MAIN.M10.nRawEncoderULINT <-> FB Inputs Channel 1/Position
//   txi_optics Instance <-> Device 1 (EtherCAT)/Term 1 (EK1200)/Term 6 (EK1122)/EK1100_M2K3/EL5042_M2K3_Xupdwn
//     PlcTask Inputs/MAIN.M2K3.fbRunHOMS.stXdwnEnc/Count <-> FB Inputs Channel 2/Position
//     PlcTask Inputs/MAIN.M2K3.fbRunHOMS.stXupEnc/Count <-> FB Inputs Channel 1/Position
//     PlcTask Inputs/MAIN.M8.nRawEncoderULINT <-> FB Inputs Channel 1/Position
//     PlcTask Inputs/MAIN.M9.nRawEncoderULINT <-> FB Inputs Channel 2/Position
//   txi_optics Instance <-> Device 1 (EtherCAT)/Term 1 (EK1200)/Term 6 (EK1122)/EK1100_M2K3/EL5042_M2K3_Yupdwn
//     PlcTask Inputs/MAIN.M2K3.fbRunHOMS.stYdwnEnc/Count <-> FB Inputs Channel 2/Position
//     PlcTask Inputs/MAIN.M2K3.fbRunHOMS.stYupEnc/Count <-> FB Inputs Channel 1/Position
//     PlcTask Inputs/MAIN.M6.nRawEncoderULINT <-> FB Inputs Channel 1/Position
//     PlcTask Inputs/PRG_MR2K3_SOMS.bMR2K3_Y_ENC_Ready <-> FB Inputs Channel 1/Status/Ready
//     PlcTask Inputs/PRG_MR2K3_SOMS.bMR2K3_Y_ENC_TxPDO <-> FB Inputs Channel 1/Status/TxPDO State
//   txi_optics Instance <-> Device 1 (EtherCAT)/Term 1 (EK1200)/Term 6 (EK1122)/EK1100_M2K3/EL6001_M2K3_PitchFine
//     SerialIO Inputs/GVL_SerialIO.Serial_stComIn_M2K3/D[{0..21}] <-> COM Inputs/Data In {0..21}  (22 links)
//     SerialIO Inputs/GVL_SerialIO.Serial_stComIn_M2K3/Status <-> COM Inputs/Status
//     SerialIO Outputs/GVL_SerialIO.Serial_stComOut_M2K3/Ctrl <-> COM Outputs/Ctrl
//     SerialIO Outputs/GVL_SerialIO.Serial_stComOut_M2K3/D[{0..21}] <-> COM Outputs/Data Out {0..21}  (22 links)
//   txi_optics Instance <-> Device 1 (EtherCAT)/Term 1 (EK1200)/Term 6 (EK1122)/EK1100_M2K3/EL7047_M2K3_PitchCoarse
//     PlcTask Inputs/MAIN.M10.bLimitBackwardEnable <-> STM Status/Status/Digital input 2
//     PlcTask Inputs/MAIN.M10.bLimitForwardEnable <-> STM Status/Status/Digital input 1
//   txi_optics Instance <-> Device 1 (EtherCAT)/Term 1 (EK1200)/Term 6 (EK1122)/EK1100_M2K3/EL7047_M2K3_Xdwn
//     PlcTask Inputs/MAIN.M9.bLimitBackwardEnable <-> STM Status/Status/Digital input 2
//     PlcTask Inputs/MAIN.M9.bLimitForwardEnable <-> STM Status/Status/Digital input 1
//   txi_optics Instance <-> Device 1 (EtherCAT)/Term 1 (EK1200)/Term 6 (EK1122)/EK1100_M2K3/EL7047_M2K3_Xup
//     PlcTask Inputs/MAIN.M8.bLimitBackwardEnable <-> STM Status/Status/Digital input 2
//     PlcTask Inputs/MAIN.M8.bLimitForwardEnable <-> STM Status/Status/Digital input 1
//   txi_optics Instance <-> Device 1 (EtherCAT)/Term 1 (EK1200)/Term 6 (EK1122)/EK1100_M2K3/EL7047_M2K3_Ydwn
//     PlcTask Inputs/MAIN.M7.bLimitBackwardEnable <-> STM Status/Status/Digital input 2
//     PlcTask Inputs/MAIN.M7.bLimitForwardEnable <-> STM Status/Status/Digital input 1
//   txi_optics Instance <-> Device 1 (EtherCAT)/Term 1 (EK1200)/Term 6 (EK1122)/EK1100_M2K3/EL7047_M2K3_Yup
//     PlcTask Inputs/MAIN.M6.bLimitBackwardEnable <-> STM Status/Status/Digital input 2
//     PlcTask Inputs/MAIN.M6.bLimitForwardEnable <-> STM Status/Status/Digital input 1
//   txi_optics Instance <-> NC-Task 1 SAF/Axes/M1K3-Pitch
//     PlcTask Inputs/MAIN.M5.Axis.NcToPlc <-> Outputs/ToPlc
//     PlcTask Outputs/MAIN.M5.Axis.PlcToNc <-> Inputs/FromPlc
//   txi_optics Instance <-> NC-Task 1 SAF/Axes/M1K3-Xdwn
//     PlcTask Inputs/MAIN.M4.Axis.NcToPlc <-> Outputs/ToPlc
//     PlcTask Outputs/MAIN.M4.Axis.PlcToNc <-> Inputs/FromPlc
//   txi_optics Instance <-> NC-Task 1 SAF/Axes/M1K3-Xup
//     PlcTask Inputs/MAIN.M3.Axis.NcToPlc <-> Outputs/ToPlc
//     PlcTask Outputs/MAIN.M3.Axis.PlcToNc <-> Inputs/FromPlc
//   txi_optics Instance <-> NC-Task 1 SAF/Axes/M1K3-Ydwn
//     PlcTask Inputs/MAIN.M2.Axis.NcToPlc <-> Outputs/ToPlc
//     PlcTask Outputs/MAIN.M2.Axis.PlcToNc <-> Inputs/FromPlc
//   txi_optics Instance <-> NC-Task 1 SAF/Axes/M1K3-Yup
//     PlcTask Inputs/MAIN.M1.Axis.NcToPlc <-> Outputs/ToPlc
//     PlcTask Outputs/MAIN.M1.Axis.PlcToNc <-> Inputs/FromPlc
//   txi_optics Instance <-> NC-Task 1 SAF/Axes/M2K3-Pitch
//     PlcTask Inputs/MAIN.M10.Axis.NcToPlc <-> Outputs/ToPlc
//     PlcTask Outputs/MAIN.M10.Axis.PlcToNc <-> Inputs/FromPlc
//   txi_optics Instance <-> NC-Task 1 SAF/Axes/M2K3-Xdwn
//     PlcTask Inputs/MAIN.M9.Axis.NcToPlc <-> Outputs/ToPlc
//     PlcTask Outputs/MAIN.M9.Axis.PlcToNc <-> Inputs/FromPlc
//   txi_optics Instance <-> NC-Task 1 SAF/Axes/M2K3-Xup
//     PlcTask Inputs/MAIN.M8.Axis.NcToPlc <-> Outputs/ToPlc
//     PlcTask Outputs/MAIN.M8.Axis.PlcToNc <-> Inputs/FromPlc
//   txi_optics Instance <-> NC-Task 1 SAF/Axes/M2K3-Ydwn
//     PlcTask Inputs/MAIN.M7.Axis.NcToPlc <-> Outputs/ToPlc
//     PlcTask Outputs/MAIN.M7.Axis.PlcToNc <-> Inputs/FromPlc
//   txi_optics Instance <-> NC-Task 1 SAF/Axes/M2K3-Yup
//     PlcTask Inputs/MAIN.M6.Axis.NcToPlc <-> Outputs/ToPlc
//     PlcTask Outputs/MAIN.M6.Axis.PlcToNc <-> Inputs/FromPlc

CONFIGURATION txi_optics
    RESOURCE PLC ON TwinCAT3
        TASK PiezoDriver(INTERVAL := T#1ms, PRIORITY := 3);
        TASK PlcTask(INTERVAL := T#10ms, PRIORITY := 20);
        TASK SerialIO(INTERVAL := T#2ms, PRIORITY := 1);
        PROGRAM PiezoSerial WITH PiezoDriver : PiezoSerial;
        PROGRAM MAIN WITH PlcTask : MAIN;
        PROGRAM P_Serial_Com WITH SerialIO : P_Serial_Com;
    END_RESOURCE
END_CONFIGURATION

// ---- GVLs/GVL_COM_Buffers.TcGVL
VAR_GLOBAL
    // M1K3
    Serial_RXBuffer_M1K3 : ComBuffer;
    Serial_TXBuffer_M1K3 : ComBuffer;

    // M2K3
    Serial_RXBuffer_M2K3 : ComBuffer;
    Serial_TXBuffer_M2K3 : ComBuffer;
END_VAR

// ---- Version/Global_Version.TcGVL
{attribute 'TcGenerated'}
{attribute 'no-analysis'}
{attribute 'linkalways'}
// This function has been automatically generated from the project information.
VAR_GLOBAL CONSTANT
    {attribute 'const_non_replaced'}
    stLibVersion_lcls_plc_txi_optics : ST_LibVersion := (iMajor := 0, iMinor := 2, iBuild := 0, iRevision := 0, nFlags := 1, sVersion := '0.2.0');
END_VAR

// ---- GVLs/GVL_M1K3.TcGVL
{attribute 'qualified_only'}
VAR_GLOBAL
    // Pitch Mechanism:
    {attribute 'TcLinkTo' := '.diEncCnt:=TIIB[EL5042_M1K3_Pitch]^FB Inputs Channel 1^Position'}
    M1K3_Pitch : HOMS_PitchMechanism := (ReqPosLimHi := 1,
                                         ReqPosLimLo := -1,
                                         diEncPosLimHi := 1,
                                         diEncPosLimLo := -1);
END_VAR

// ---- GVLs/GVL_M1K3_Constants.TcGVL
{attribute 'qualified_only'}
VAR_GLOBAL CONSTANT
    // Encoder reference values in counts = nm
    // Enc Ref Vals from FAT
    nYUP_ENC_REF : ULINT := 108743550;
    nYDWN_ENC_REF : ULINT := 108243370;
    nXUP_ENC_REF : ULINT := 19628100;
    nXDWN_ENC_REF : ULINT := 20865800;
END_VAR

// ---- GVLs/GVL_M2K3.TcGVL
{attribute 'qualified_only'}
VAR_GLOBAL
    // Pitch Mechanism
    {attribute 'TcLinkTo' := '.diEncCnt:=TIIB[EL5042_M2K3_Pitch]^FB Inputs Channel 1^Position'}
    M2K3_Pitch : HOMS_PitchMechanism := (ReqPosLimHi := 58900,
                                         ReqPosLimLo := 57500,
                                         diEncPosLimHi := 10602000,
                                         diEncPosLimLo := 10350000);
END_VAR

// ---- GVLs/GVL_M2K3_Constants.TcGVL
{attribute 'qualified_only'}
VAR_GLOBAL CONSTANT
    // Encoder reference values in counts = nm
    // Enc Ref Vals after realignment with metrology
    nYUP_ENC_REF : ULINT := 40653120;
    nYDWN_ENC_REF : ULINT := 43456180;
    nXUP_ENC_REF : ULINT := 23635520;
    nXDWN_ENC_REF : ULINT := 22541650;
END_VAR

// ---- GVLs/GVL_PMPS.TcGVL
{attribute 'qualified_only'}
VAR_GLOBAL
    {attribute 'pytmc' := 'pv: PLC:TXI:KFE:OPTICS:ARB:01'}
    fbArbiter1: FB_Arbiter(1);
    {attribute 'pytmc' := 'pv: PLC:TXI:KFE:OPTICS:ARB:02'}
    fbArbiter2: FB_Arbiter(2);
    {attribute 'pytmc' := 'pv: PLC:TXI:KFE:OPTICS:FFO:01'}
    {attribute 'TcLinkTo' := '.q_xFastFaultOut:=TIIB[PMPS_PRE]^IO Outputs^FFO'}
    fbFastFaultOutput1: FB_HardwareFFOutput := (bAutoReset := TRUE , i_sNetID:='172.21.42.126.1.1' );
END_VAR

// ---- GVLs/GVL_SerialIO.TcGVL
VAR_GLOBAL
    //Better have your inputs and outputs!
    // M1K3
    Serial_stComIn_M1K3   AT %I*	:	EL6inData22B (*KL6inData22B*);
    Serial_stComOut_M1K3  AT %Q*	:	EL6outData22B (*KL6outData22B*);

    // M2L0
    Serial_stComIn_M2K3   AT %I*	:	EL6inData22B (*KL6inData22B*);
    Serial_stComOut_M2K3  AT %Q*	:	EL6outData22B (*KL6outData22B*);
END_VAR

// ---- POUs/Serial Comm/PiezoSerial.TcPOU
PROGRAM PiezoSerial
VAR
    //PI Serial
    fbE621SerialDriver_M1K3 : FB_PI_E621_SerialDriver;
    rtInitParams_M1K3	:	R_TRIG;
    tonTimeoutRst_M1K3	: TON := (PT:=T#2S); //For timeout reset

    fbE621SerialDriver_M2K3 : FB_PI_E621_SerialDriver;
    rtInitParams_M2K3	:	R_TRIG;
    tonTimeoutRst_M2K3	: TON := (PT:=T#2S); //For timeout reset
END_VAR

//Piezo E-621
///////////////////////
fbE621SerialDriver_M1K3.i_xExecute := TRUE;
fbE621SerialDriver_M1K3.i_xExecute R= fbE621SerialDriver_M1K3.q_xDone;
fbE621SerialDriver_M1K3(iq_stPiezoAxis:= GVL_M1K3.M1K3_Pitch.Piezo,
                        iq_stSerialRXBuffer:= Serial_RXBuffer_M1K3,
                        iq_stSerialTXBuffer:= Serial_TXBuffer_M1K3);

fbE621SerialDriver_M2K3.i_xExecute := TRUE;
fbE621SerialDriver_M2K3.i_xExecute R= fbE621SerialDriver_M2K3.q_xDone;
fbE621SerialDriver_M2K3(iq_stPiezoAxis:= GVL_M2K3.M2K3_Pitch.Piezo,
                        iq_stSerialRXBuffer:= Serial_RXBuffer_M2K3,
                        iq_stSerialTXBuffer:= Serial_TXBuffer_M2K3);

END_PROGRAM

// ---- POUs/MAIN.TcPOU
PROGRAM MAIN
VAR
    // M1K3
    // Motors
    {attribute 'TcLinkTo' := '.bLimitForwardEnable:=TIIB[EL7047_M1K3_Yup]^STM Status^Status^Digital input 1;
                              .bLimitBackwardEnable:=TIIB[EL7047_M1K3_Yup]^STM Status^Status^Digital input 2;
                              .nRawEncoderULINT:=TIIB[EL5042_M1K3_Yupdwn]^FB Inputs Channel 1^Position'}
    {attribute 'pytmc' := '
        pv: MR1K3:SOMS:MMS:YUP
    '}
    M1 : DUT_MotionStage := (fVelocity:=100.0, nEnableMode:=ENUM_StageEnableMode.ALWAYS,  bPowerSelf:=True); // M1K3 Yup
    fbMotionStage_m1 : FB_MotionStage;

    {attribute 'TcLinkTo' := '.bLimitForwardEnable:=TIIB[EL7047_M1K3_Ydwn]^STM Status^Status^Digital input 1;
                              .bLimitBackwardEnable:=TIIB[EL7047_M1K3_Ydwn]^STM Status^Status^Digital input 2'}
    {attribute 'pytmc' := '
        pv: MR1K3:SOMS:MMS:YDWN
    '}
    M2 : DUT_MotionStage := (fVelocity:=100.0, nEnableMode:=ENUM_StageEnableMode.ALWAYS,  bPowerSelf:=True); // M1K3 Ydwn
    fbMotionStage_m2 : FB_MotionStage;

    {attribute 'TcLinkTo' := '.bLimitForwardEnable:=TIIB[EL7047_M1K3_Xup]^STM Status^Status^Digital input 1;
                              .bLimitBackwardEnable:=TIIB[EL7047_M1K3_Xup]^STM Status^Status^Digital input 2;
                              .nRawEncoderULINT:=TIIB[EL5042_M1K3_Xupdwn]^FB Inputs Channel 1^Position'}
    {attribute 'pytmc' := '
        pv: MR1K3:SOMS:MMS:XUP
    '}
    M3 : DUT_MotionStage := (fVelocity:=300.0, nEnableMode:=ENUM_StageEnableMode.ALWAYS,  bPowerSelf:=True); // M1K3 Xup
    fbMotionStage_m3 : FB_MotionStage;

    {attribute 'TcLinkTo' := '.bLimitForwardEnable:=TIIB[EL7047_M1K3_Xdwn]^STM Status^Status^Digital input 1;
                              .bLimitBackwardEnable:=TIIB[EL7047_M1K3_Xdwn]^STM Status^Status^Digital input 2;
                              .nRawEncoderULINT:=TIIB[EL5042_M1K3_Xupdwn]^FB Inputs Channel 2^Position'}
    {attribute 'pytmc' := '
        pv: MR1K3:SOMS:MMS:XDWN
    '}
    M4 : DUT_MotionStage := (fVelocity:=300.0, nEnableMode:=ENUM_StageEnableMode.ALWAYS,  bPowerSelf:=True); // M1K3 Xdwn
    fbMotionStage_m4 : FB_MotionStage;

    {attribute 'TcLinkTo' := '.bLimitForwardEnable:=TIIB[EL7047_M1K3_PitchCoarse]^STM Status^Status^Digital input 1;
                              .bLimitBackwardEnable:=TIIB[EL7047_M1K3_PitchCoarse]^STM Status^Status^Digital input 2;
                              .nRawEncoderULINT:=TIIB[EL5042_M1K3_Pitch]^FB Inputs Channel 1^Position'}
    {attribute 'pytmc' := '
        pv: MR1K3:SOMS:MMS:PITCH
    '}
    M5 : DUT_MotionStage := (fVelocity:=50.0,  bPowerSelf:=True); // M1K3 Pitch Stepper

    {attribute 'TcLinkTo' := '.fbRunHOMS.bSTOEnable1:=TIIB[EL1004_M1K3_STO]^Channel 1^Input;
                              .fbRunHOMS.bSTOEnable2:=TIIB[EL1004_M1K3_STO]^Channel 2^Input;
                              .fbRunHOMS.stYupEnc.Count:=TIIB[EL5042_M1K3_Yupdwn]^FB Inputs Channel 1^Position;
                              .fbRunHOMS.stYdwnEnc.Count:=TIIB[EL5042_M1K3_Yupdwn]^FB Inputs Channel 2^Position;
                              .fbRunHOMS.stXupEnc.Count:=TIIB[EL5042_M1K3_Xupdwn]^FB Inputs Channel 1^Position;
                              .fbRunHOMS.stXdwnEnc.Count:=TIIB[EL5042_M1K3_Xupdwn]^FB Inputs Channel 2^Position'}
    {attribute 'pytmc' := '
        pv: MR1K3:SOMS
    '}
    M1K3 : DUT_HOMS;

    // Encoder Arrays/RMS Watch:
    {attribute 'pytmc' := '
        pv: MR1K3:SOMS:ENC:Y
    '}
    fbYRMSErrorM1K3 : FB_RMSWatch;
    fMaxYRMSErrorM1K3 : LREAL;
    fMinYRMSErrorM1K3 : LREAL;

    {attribute 'pytmc' := '
        pv: MR1K3:SOMS:ENC:X
    '}
    fbXRMSErrorM1K3 : FB_RMSWatch;
    fMaxXRMSErrorM1K3 : LREAL;
    fMinXRMSErrorM1K3 : LREAL;

    {attribute 'pytmc' := '
        pv: MR1K3:SOMS:ENC:PITCH
    '}
    fbPitchRMSErrorM1K3 : FB_RMSWatch;
    fMaxPitchRMSErrorM1K3 : LREAL;
    fMinPitchRMSErrorM1K3 : LREAL;

    // Pitch Control
    fbM1K3PitchControl : FB_PitchControl;
    bM1K3PitchDone : BOOL;
    bM1K3PitchBusy : BOOL;

    {attribute 'TcLinkTo' := 'TIIB[EL2004_M1K3_VCV]^Channel 1^Output'}
    {attribute 'pytmc' := '
        pv: MR1K3:SOMS:VCV
        io: io
        field: ZNAM OFF
        field: ONAM ON
    '}
    bActivateVarCoolMR1K3 AT %Q* : BOOL;


    // M2K3
    // Motors
    {attribute 'TcLinkTo' := '.bLimitForwardEnable:=TIIB[EL7047_M2K3_Yup]^STM Status^Status^Digital input 1;
                              .bLimitBackwardEnable:=TIIB[EL7047_M2K3_Yup]^STM Status^Status^Digital input 2;
                              .nRawEncoderULINT:=TIIB[EL5042_M2K3_Yupdwn]^FB Inputs Channel 1^Position'}
    {attribute 'pytmc' := '
        pv: MR2K3:SOMS:MMS:YUP
    '}
    M6 : DUT_MotionStage := (fVelocity:=100.0, nEnableMode:=ENUM_StageEnableMode.ALWAYS,  bPowerSelf:=True); // M2K3 Yup
    fbMotionStage_m6 : FB_MotionStage;

    {attribute 'TcLinkTo' := '.bLimitForwardEnable:=TIIB[EL7047_M2K3_Ydwn]^STM Status^Status^Digital input 1;
                              .bLimitBackwardEnable:=TIIB[EL7047_M2K3_Ydwn]^STM Status^Status^Digital input 2'}
    {attribute 'pytmc' := '
        pv: MR2K3:SOMS:MMS:YDWN
    '}
    M7 : DUT_MotionStage := (fVelocity:=100.0, nEnableMode:=ENUM_StageEnableMode.ALWAYS,  bPowerSelf:=True); // M2K3 Ydwn
    fbMotionStage_m7 : FB_MotionStage;

    {attribute 'TcLinkTo' := '.bLimitForwardEnable:=TIIB[EL7047_M2K3_Xup]^STM Status^Status^Digital input 1;
                              .bLimitBackwardEnable:=TIIB[EL7047_M2K3_Xup]^STM Status^Status^Digital input 2;
                              .nRawEncoderULINT:=TIIB[EL5042_M2K3_Xupdwn]^FB Inputs Channel 1^Position'}
    {attribute 'pytmc' := '
        pv: MR2K3:SOMS:MMS:XUP
    '}
    M8 : DUT_MotionStage := (fVelocity:=150.0, nEnableMode:=ENUM_StageEnableMode.ALWAYS,  bPowerSelf:=True); // M2K3 Xup
    fbMotionStage_m8 : FB_MotionStage;

    {attribute 'TcLinkTo' := '.bLimitForwardEnable:=TIIB[EL7047_M2K3_Xdwn]^STM Status^Status^Digital input 1;
                              .bLimitBackwardEnable:=TIIB[EL7047_M2K3_Xdwn]^STM Status^Status^Digital input 2;
                              .nRawEncoderULINT:=TIIB[EL5042_M2K3_Xupdwn]^FB Inputs Channel 2^Position'}
    {attribute 'pytmc' := '
        pv: MR2K3:SOMS:MMS:XDWN
    '}
    M9 : DUT_MotionStage := (fVelocity:=150.0, nEnableMode:=ENUM_StageEnableMode.ALWAYS,  bPowerSelf:=True); // M2K3 Xdwn
    fbMotionStage_m9 : FB_MotionStage;

    {attribute 'TcLinkTo' := '.bLimitForwardEnable:=TIIB[EL7047_M2K3_PitchCoarse]^STM Status^Status^Digital input 1;
                              .bLimitBackwardEnable:=TIIB[EL7047_M2K3_PitchCoarse]^STM Status^Status^Digital input 2;
                              .nRawEncoderULINT:=TIIB[EL5042_M2K3_Pitch]^FB Inputs Channel 1^Position'}
    {attribute 'pytmc' := '
        pv: MR2K3:SOMS:MMS:PITCH
    '}
    M10 : DUT_MotionStage := (fVelocity:=50.0, nEnableMode:=ENUM_StageEnableMode.ALWAYS,  bPowerSelf:=True); // M2K3 Pitch Stepper

    {attribute 'TcLinkTo' := '.fbRunHOMS.bSTOEnable1:=TIIB[EL1004_M2K3_STO]^Channel 1^Input;
                              .fbRunHOMS.bSTOEnable2:=TIIB[EL1004_M2K3_STO]^Channel 2^Input;
                              .fbRunHOMS.stYupEnc.Count:=TIIB[EL5042_M2K3_Yupdwn]^FB Inputs Channel 1^Position;
                              .fbRunHOMS.stYdwnEnc.Count:=TIIB[EL5042_M2K3_Yupdwn]^FB Inputs Channel 2^Position;
                              .fbRunHOMS.stXupEnc.Count:=TIIB[EL5042_M2K3_Xupdwn]^FB Inputs Channel 1^Position;
                              .fbRunHOMS.stXdwnEnc.Count:=TIIB[EL5042_M2K3_Xupdwn]^FB Inputs Channel 2^Position'}
    {attribute 'pytmc' := '
        pv: MR2K3:SOMS
    '}
    M2K3 : DUT_HOMS;

    // Encoder Arrays/RMS Watch:
    {attribute 'pytmc' := '
        pv: MR2K3:SOMS:ENC:Y
    '}
    fbYRMSErrorM2K3 : FB_RMSWatch;
    fMaxYRMSErrorM2K3 : LREAL;
    fMinYRMSErrorM2K3 : LREAL;

    {attribute 'pytmc' := '
        pv: MR2K3:SOMS:ENC:X
    '}
    fbXRMSErrorM2K3 : FB_RMSWatch;
    fMaxXRMSErrorM2K3 : LREAL;
    fMinXRMSErrorM2K3 : LREAL;

    {attribute 'pytmc' := '
        pv: MR2K3:SOMS:ENC:PITCH
    '}
    fbPitchRMSErrorM2K3 : FB_RMSWatch;
    fMaxPitchRMSErrorM2K3 : LREAL;
    fMinPitchRMSErrorM2K3 : LREAL;

    // Pitch Control
    fbM2K3PitchControl : FB_PitchControl;
    bM2K3PitchDone : BOOL;
    bM2K3PitchBusy : BOOL;

    // Lost serial comm to E621 controller, unsure why...
    fbMotionStage_m10 : FB_MotionStage;

    {attribute 'TcLinkTo' := 'TIIB[EL2004_M2K3_VCV]^Channel 1^Output'}
    {attribute 'pytmc' := '
        pv: MR2K3:SOMS:VCV
        io: io
        field: ZNAM OFF
        field: ONAM ON
    '}
    bActivateVarCoolMR2K3 AT %Q* : BOOL;

     // MR1K3 Flow Press Sensors
    {attribute 'TcLinkTo' := '.fbFlow_1.iRaw := TIIB[EL3054_M1K3_FWM_PRSM]^AI Standard Channel 1^Value;
                                 .fbFlow_2.iRaw := TIIB[EL3054_M1K3_FWM_PRSM]^AI Standard Channel 2^Value;
                              .fbPress_1.iRaw := TIIB[EL3054_M1K3_FWM_PRSM]^AI Standard Channel 3^Value
    '}
    {attribute 'pytmc' := '
        pv: MR1K3:SOMS
    '}
    fbCoolingPanelMR1K3 : FB_Axilon_Cooling_2f1p;

    // MR2K3 Flow Press Sensors
    {attribute 'TcLinkTo' := '.fbFlow_1.iRaw := TIIB[EL3054_M2K3_FWM_PRSM]^AI Standard Channel 1^Value;
                                 .fbFlow_2.iRaw := TIIB[EL3054_M2K3_FWM_PRSM]^AI Standard Channel 2^Value;
                              .fbPress_1.iRaw := TIIB[EL3054_M2K3_FWM_PRSM]^AI Standard Channel 3^Value
    '}
    {attribute 'pytmc' := '
        pv: MR2K3:SOMS
    '}
    fbCoolingPanelMR2K3 : FB_Axilon_Cooling_2f1p;
END_VAR

// M1K3
M1K3.fbRunHOMS(stYup:=M1,
               stYdwn:=M2,
               stXup:=M3,
               stXdwn:=M4,
               stPitch:=M5,
               nYupEncRef:=GVL_M1K3_Constants.nYUP_ENC_REF,
               nYdwnEncRef:=GVL_M1K3_Constants.nYDWN_ENC_REF,
               nXupEncRef:=GVL_M1K3_Constants.nXUP_ENC_REF,
               nXdwnEncRef:=GVL_M1K3_Constants.nXDWN_ENC_REF,
               bExecuteCoupleY:=M1K3.bExecuteCoupleY,
               bExecuteCoupleX:=M1K3.bExecuteCoupleX,
               bExecuteDecoupleY:=M1K3.bExecuteDecoupleY,
               bExecuteDecoupleX:=M1K3.bExecuteDecoupleX,
               bGantryAlreadyCoupledY=>M1K3.bGantryAlreadyCoupledY,
               bGantryAlreadyCoupledX=>M1K3.bGantryAlreadyCoupledX,
               nCurrGantryY=>M1K3.nCurrGantryY,
               nCurrGantryX=>M1K3.nCurrGantryX);

// Convert nCurrGantry to um (smaller number) to read out in epics
M1K3.fCurrGantryY_um := LINT_TO_REAL(M1K3.nCurrGantryY) / 1000.0;
M1K3.fCurrGantryX_um := LINT_TO_REAL(M1K3.nCurrGantryX) / 1000.0;

// FB_MotionStage's for non-piezo axes
fbMotionStage_m1(stMotionStage:=M1);
fbMotionStage_m2(stMotionStage:=M2);
fbMotionStage_m3(stMotionStage:=M3);
fbMotionStage_m4(stMotionStage:=M4);

// Calculate Pitch RMS Error:
fbYRMSErrorM1K3(stMotionStage:=M1,
                fMaxRMSError=>fMaxYRMSErrorM1K3,
                fMinRMSError=>fMinYRMSErrorM1K3);

fbXRMSErrorM1K3(stMotionStage:=M3,
                fMaxRMSError=>fMaxXRMSErrorM1K3,
                fMinRMSError=>fMinXRMSErrorM1K3);

fbPitchRMSErrorM1K3(stMotionStage:=M5,
                    fMaxRMSError=>fMaxPitchRMSErrorM1K3,
                    fMinRMSError=>fMinPitchRMSErrorM1K3);

// Pitch Control
fbM1K3PitchControl(Pitch:=GVL_M1K3.M1K3_Pitch,
                   Stepper:=M5,
                   lrCurrentSetpoint:=M5.fPosition,
                   q_bDone=>bM1K3PitchDone,
                   q_bBusy=>bM1K3PitchBusy);
// When STO hit, need to reset SP
IF NOT M5.bHardwareEnable THEN
    M5.fPosition := M5.stAxisStatus.fActPosition;
END_IF

// M2K3
M2K3.fbRunHOMS(stYup:=M6,
               stYdwn:=M7,
               stXup:=M8,
               stXdwn:=M9,
               stPitch:=M10,
               nYupEncRef:=GVL_M2K3_Constants.nYUP_ENC_REF,
               nYdwnEncRef:=GVL_M2K3_Constants.nYDWN_ENC_REF,
               nXupEncRef:=GVL_M2K3_Constants.nXUP_ENC_REF,
               nXdwnEncRef:=GVL_M2K3_Constants.nXDWN_ENC_REF,
               bExecuteCoupleY:=M2K3.bExecuteCoupleY,
               bExecuteCoupleX:=M2K3.bExecuteCoupleX,
               bExecuteDecoupleY:=M2K3.bExecuteDecoupleY,
               bExecuteDecoupleX:=M2K3.bExecuteDecoupleX,
               bGantryAlreadyCoupledY=>M2K3.bGantryAlreadyCoupledY,
               bGantryAlreadyCoupledX=>M2K3.bGantryAlreadyCoupledX,
               nCurrGantryY=>M2K3.nCurrGantryY,
               nCurrGantryX=>M2K3.nCurrGantryX);

// Convert nCurrGantry to um (smaller number) to read out in epics
M2K3.fCurrGantryY_um := LINT_TO_REAL(M2K3.nCurrGantryY) / 1000;
M2K3.fCurrGantryX_um := LINT_TO_REAL(M2K3.nCurrGantryX) / 1000;

// FB_MotionStage's for non-piezo axes
fbMotionStage_m6(stMotionStage:=M6);
fbMotionStage_m7(stMotionStage:=M7);
fbMotionStage_m8(stMotionStage:=M8);
fbMotionStage_m9(stMotionStage:=M9);

// Calculate RMS Error:
fbYRMSErrorM2K3(stMotionStage:=M6,
                fMaxRMSError=>fMaxYRMSErrorM2K3,
                fMinRMSError=>fMinYRMSErrorM2K3);

fbXRMSErrorM2K3(stMotionStage:=M8,
                fMaxRMSError=>fMaxXRMSErrorM2K3,
                fMinRMSError=>fMinXRMSErrorM2K3);

fbPitchRMSErrorM2K3(stMotionStage:=M10,
                    fMaxRMSError=>fMaxPitchRMSErrorM2K3,
                    fMinRMSError=>fMinPitchRMSErrorM2K3);

(*
3-15-20: Lost serial comm with E621 controller, unsure why....
// Pitch Control
fbM2K3PitchControl(Pitch:=GVL_M2K3.M2K3_Pitch,
                   Stepper:=M10,
                   lrCurrentSetpoint:=M10.fPosition,
                   q_bDone=>bM2K3PitchDone,
                   q_bBusy=>bM2K3PitchBusy);
// When STO hit, need to reset SP
IF NOT M10.bHardwareEnable THEN
    M10.fPosition := M10.stAxisStatus.fActPosition;
END_IF
*)
fbMotionStage_m10(stMotionStage:=M10);

// MR1K3 Flow Pressure Sensors
fbCoolingPanelMR1K3();
fbCoolingPanelMR2K3();
PRG_1_PlcTask();

END_PROGRAM

// ---- POUs/PRG_1_PlcTask.TcPOU
PROGRAM PRG_1_PlcTask
VAR
END_VAR

PRG_2_PMPS_POST();
PRG_MR1K3_SOMS();
PRG_MR2K3_SOMS();

END_PROGRAM

// ---- POUs/PRG_2_PMPS_POST.TcPOU
PROGRAM PRG_2_PMPS_POST
VAR
    fbArbiterIO: FB_SubSysToArbiter_IO;
    fb_vetoArbiter: FB_VetoArbiter;
END_VAR


GVL_PMPS.fbFastFaultOutput1.Execute();

fbArbiterIO(
    Arbiter:=GVL_PMPS.fbArbiter1,
    fbFFHWO:=GVL_PMPS.fbFastFaultOutput1);
//Arb2 in hutch
(**fb_vetoArbiter(bVeto:= PMPS_GVL.stCurrentBeamParameters.aVetoDevices[PMPS.L_Stopper.ST1L1],
                HigherAuthority := GVL_PMPS.fbArbiter1,
                LowerAuthority := GVL_PMPS.fbArbiter2,
                FFO := GVL_PMPS.fbFastFaultOutput1);
**)
//ff2_ff1_link_optics(
    //io_fbFFHWO := GVL_PMPS.fbFastFaultOutput1,
    //i_xOK :=  GVL_PMPS.fbFastFaultOutput2.q_xFastFaultOut);

//Code for Removing arbitration
GVL_PMPS.fbArbiter1.AddRequest(nReqID := 49, stReqBp := PMPS_GVL.cstFullBeam, sDevName := 'txi-kfe-optics');
GVL_PMPS.fbArbiter2.AddRequest(nReqID := 50, stReqBp := PMPS_GVL.cstFullBeam, sDevName := 'txi-kfe-optics');

//send encoder values for veto

END_PROGRAM

// ---- POUs/PRG_MR1K3_SOMS.TcPOU
PROGRAM PRG_MR1K3_SOMS
VAR
    {attribute 'TcLinkTo' := 'TIIB[PMPS_PRE]^IO Outputs^MR1K3_Y_ENC'}
    nMR1K3_Y_ENC_PMPS AT %Q* : ULINT;
    {attribute 'TcLinkTo' := 'TIIB[EL5042_M1K3_Yupdwn]^FB Inputs Channel 1^Status^Ready'}
    bMR1K3_Y_ENC_Ready AT %I* : BOOL;
    {attribute 'TcLinkTo' := 'TIIB[EL5042_M1K3_Yupdwn]^FB Inputs Channel 1^Status^TxPDO State'}
    bMR1K3_Y_ENC_TxPDO AT %I* : BOOL;
END_VAR

nMR1K3_Y_ENC_PMPS := MAIN.M1.nRawEncoderULINT;

END_PROGRAM

// ---- POUs/PRG_MR2K3_SOMS.TcPOU
PROGRAM PRG_MR2K3_SOMS
VAR
    {attribute 'TcLinkTo' := 'TIIB[PMPS_PRE]^IO Outputs^MR2K3_Y_ENC'}
    nMR2K3_Y_ENC_PMPS AT %Q* : ULINT;
    {attribute 'TcLinkTo' := 'TIIB[EL5042_M2K3_Yupdwn]^FB Inputs Channel 1^Status^Ready'}
    bMR2K3_Y_ENC_Ready AT %I* : BOOL;
    {attribute 'TcLinkTo' := 'TIIB[EL5042_M2K3_Yupdwn]^FB Inputs Channel 1^Status^TxPDO State'}
    bMR2K3_Y_ENC_TxPDO AT %I* : BOOL;
END_VAR

nMR2K3_Y_ENC_PMPS := MAIN.M6.nRawEncoderULINT;

END_PROGRAM

// ---- POUs/Serial Comm/P_Serial_Com.TcPOU
PROGRAM P_Serial_Com
VAR
    fbSerialLineControl_EL6001_M1K3: SerialLineControl;
    fbSerialLineControl_EL6001_M2K3: SerialLineControl;
END_VAR

//These are the global IOs...don't forget to copy your data into them

(* EL6001 Serial port 0 com function *)
fbSerialLineControl_EL6001_M1K3(Mode:= SERIALLINEMODE_EL6_22B (*SERIALLINEMODE_KL6_22B_STANDARD*),
                                pComIn:= ADR(Serial_stComIn_M1K3),
                                   pComOut:=ADR(Serial_stComOut_M1K3),
                                SizeComIn:= SIZEOF(Serial_stComIn_M1K3),
                                TxBuffer:= Serial_TXBuffer_M1K3,
                                RxBuffer:= Serial_RXBuffer_M1K3,
                                Error=> ,
                                ErrorID=> );

fbSerialLineControl_EL6001_M2K3(Mode:= SERIALLINEMODE_EL6_22B (*SERIALLINEMODE_KL6_22B_STANDARD*),
                                pComIn:= ADR(Serial_stComIn_M2K3),
                                   pComOut:=ADR(Serial_stComOut_M2K3),
                                SizeComIn:= SIZEOF(Serial_stComIn_M2K3),
                                TxBuffer:= Serial_TXBuffer_M2K3,
                                RxBuffer:= Serial_RXBuffer_M2K3,
                                Error=> ,
                                ErrorID=> );

END_PROGRAM
